// TIA Portal V16 export
// export: Created 2026-06-21T13:18:40.1372676Z, ExportSetting WithDefaults, DisplayName Totally Integrated Automation Portal, DisplayVersion V16 Update 8, DisplayName TIA Portal Version Control Interface, DisplayVersion V16 Update 8, DisplayName TIA Portal Openness, DisplayVersion V16 Update 8, DisplayName SINAMICS Startdrive Advanced, DisplayVersion V16, DisplayName SINAMICS Startdrive G130, G150, S120, S150, SINAMICS MV, S210, DisplayVersion V16, DisplayName SINAMICS Startdrive G110M, G120, G120C, G120D, G120P, DisplayVersion V16, DisplayName STEP 7 Professional, DisplayVersion V16 Update 8, DisplayName STEP 7 Safety, DisplayVersion V16 Update 7, DisplayName WinCC Advanced, DisplayVersion V16 Update 8
Screen "Motor_Control_800x480"  800x480, Number=1
  ScreenLayer 
    Circle "LMP_Run" at 341,165 size 48x48
      RangeAppearanceAnimation "RangeAppearanceAnimation"
        tag Light
        0..0: back #d9d9d9, fore #181c31
        1..1: back #00ff00, fore #181c31
    Circle "LMP_Fault" at 431,165 size 48x48
      RangeAppearanceAnimation "RangeAppearanceAnimation"
        tag Light
        0..0: back #d9d9d9, fore #181c31
        1..1: back #00ff00, fore #181c31
    Button "BTN_Start" at 226,82 size 100x45  Mode=Text, TextOff="启动", TextOn="启动"
      on Press: SetBit(Tag := Button)
      on Release: ResetBit(Tag := Button)
    Button "BTN_Reset" at 474,82 size 100x45  Mode=Text, TextOff="复位", TextOn="复位"
      on Press: SetBit(Tag := Button)
      on Release: ResetBit(Tag := Button)
    Button "BTN_Stop" at 350,82 size 100x45  Mode=Text, TextOff="停止", TextOn="停止"
      on Press: SetBit(Tag := Button)
      on Release: ResetBit(Tag := Button)
    IOField "IO_Speed" at 377,203 size 120x36  DataFormat=Decimal, FormatPattern=9999999, Mode=InOutput
    SymbolicIOField "SIO_Mode" at 377,263 size 130x36  CountVisibleItems=3, Mode=InOutput, OnValue=1, TextOff="0", TextOn="1"
    TextField "TXT_Title" at 200,20 size 400x38  Text="电机控制画面"
    TextField "TXT_ModeLabel" at 315,263 size 50x32  Text="模式"
    TextField "TXT_SpeedLabel" at 315,203 size 50x32  Text="转速"
